{attribute 'qualified_only'}
VAR_GLOBAL
	_DO 			AT%Q*:		U_OUT_IO_Translate;

END_VAR

(* stored: Version 1.1.0.1, ProductVersion 3.1.4024.10
   GVL OUT: Id {9e393b40-1de7-49b3-9092-6de105c0fc74} *)
